// TIA Portal project "AndOrLogic" (V20)

(* hardware
DEVICE "S7-1200 station_1"  S7-1200 Station
   slot 0: "Rack_0"  S7-1200 Rack  Rack  V1.0
   slot 1: "Playground_PLC"  CPU 1214C DC/DC/DC  6ES7 214-1AG40-0XB0  V4.7
   slot 3: "AQ 1x12BIT_1"  AQ1 signal board  6ES7 232-4HA30-0XB0  V1.0
*)

// ===== PLC "Playground_PLC"  CPU 1214C DC/DC/DC =====

VAR_GLOBAL   // PLC tag table "Default tag table"
   "TEST_I" AT %M0.0 : Bool;
   "TEST_O" AT %M0.1 : Bool;
END_VAR

DATA_BLOCK "INPUT"   // DB1
{ S7_Optimized_Access := 'TRUE' }
VERSION : 0.1
   VAR
      INTR_1 : Bool;
      INTR_2 : Bool;
   END_VAR
BEGIN
END_DATA_BLOCK

DATA_BLOCK "OUTPUT"   // DB2
{ S7_Optimized_Access := 'TRUE' }
VERSION : 0.1
   VAR
      LAMP : Bool;
      BUZZ : Bool;
   END_VAR
BEGIN
END_DATA_BLOCK

ORGANIZATION_BLOCK "Main"   // OB1, LAD, ProgramCycle
TITLE = "Main Program Sweep (Cycle)"
{ S7_Optimized_Access := 'TRUE' }
VERSION : 0.1
   VAR_INPUT
      Initial_Call : Bool;   // Initial call of this OB
      Remanence : Bool;   // =True, if remanent data are available
   END_VAR
BEGIN

REGION Network 1
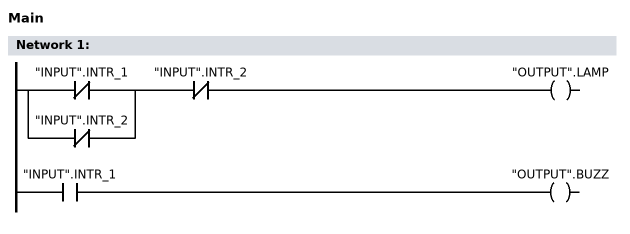
   RUNG wire#powerrail
      I_Contact( "INPUT".INTR_1 )
      wire#w1
      I_Contact( "INPUT".INTR_2 )
      Coil( "OUTPUT".LAMP )
   END_RUNG
   RUNG wire#powerrail
      I_Contact( "INPUT".INTR_2 )
   END_RUNG wire#w1
   RUNG wire#powerrail
      Contact( "INPUT".INTR_1 )
      Coil( "OUTPUT".BUZZ )
   END_RUNG
   // the same network as SCL:
   "OUTPUT".LAMP := (NOT "INPUT".INTR_1 OR NOT "INPUT".INTR_2) AND NOT "INPUT".INTR_2;
   "OUTPUT".BUZZ := "INPUT".INTR_1;
END_REGION
END_ORGANIZATION_BLOCK